// Mitsubishi GX Works2 project: 타이머2   PLC: Q02/Q02H

PROGRAM MAIN
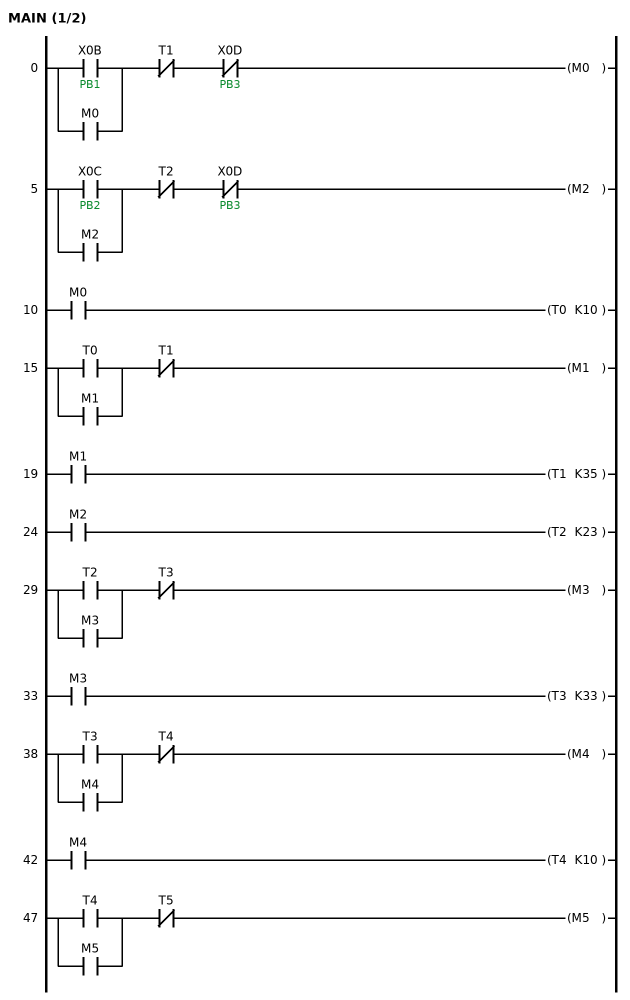
0     LD      X0B  ; PB1
      OR      M0
      ANI     T1
      ANI     X0D  ; PB3
      OUT     M0
5     LD      X0C  ; PB2
      OR      M2
      ANI     T2
      ANI     X0D  ; PB3
      OUT     M2
10    LD      M0
      OUT     T0 K10
15    LD      T0
      OR      M1
      ANI     T1
      OUT     M1
19    LD      M1
      OUT     T1 K35
24    LD      M2
      OUT     T2 K23
29    LD      T2
      OR      M3
      ANI     T3
      OUT     M3
33    LD      M3
      OUT     T3 K33
38    LD      T3
      OR      M4
      ANI     T4
      OUT     M4
42    LD      M4
      OUT     T4 K10
47    LD      T4
      OR      M5
      ANI     T5
      OUT     M5
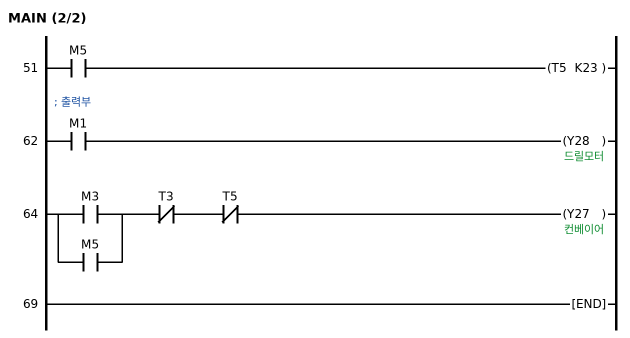
51    LD      M5
      OUT     T5 K23
; 출력부
62    LD      M1
      OUT     Y28  ; 드릴모터
64    LD      M3
      OR      M5
      ANI     T3
      ANI     T5
      OUT     Y27  ; 컨베이어
69    END
END_PROGRAM

// device comments not shown above
X0  ; 공급후진센서
X1  ; 공급전진센서
X2  ; 드릴하강센서
X3  ; 드릴상승센서
X4  ; 송출후진센서
X5  ; 송출전진센서
Y20  ; 공급전진
Y21  ; 공급후진
Y22  ; 드릴하강
Y23  ; 송출전진
Y24  ; 송출후진
